Staubli VAL3: changeOffset.pgx

public program changeOffset(num& x_nOffset[])
  local num x
  local num y
  local num z
  local point l_pPoint
  local num l_nIndex
begin
  //
  // build the pallet
  //
  // compute
  for z=0 to pEditPoint.nZ-1
    for y=0 to pEditPoint.nY-1
      for x=0 to pEditPoint.nX-1
        // set all the points
        l_pPoint=pEditPoint.tData[l_nIndex].pPoint
        l_pPoint.trsf.x=l_pPoint.trsf.x+x_nOffset*x
        l_pPoint.trsf.y=l_pPoint.trsf.y+x_nOffset[1]*y
        l_pPoint.trsf.z=l_pPoint.trsf.z+x_nOffset[2]*z
        pEditPoint.tData[l_nIndex].pPoint=l_pPoint
        l_nIndex=l_nIndex+1
      endFor
    endFor
  endFor
  //
end
